INTERFACE I_Initialise

METHOD Initialise : HRESULT
VAR_INPUT
END_VAR
END_METHOD

END_INTERFACE

(* stored: Version 1.1.0.1
   Itf I_Initialise: Id {71ff9433-60c6-4337-b06f-471ab8aac945}
   Method Initialise: Id {5f1fc26c-856c-4028-9354-4db95387c7d5} *)
